TYPE E_Servo_State :
(
    DISABLED := 0,      // motor off
    ENABLING := 10,     // turning on
    HOME_NEEDED := 15,  // on but position unknown
    HOMING := 20,       // finding home
    READY := 30,        // ready for commands
    MOVING := 40,       // moving to target
    STOPPING := 45,     // slowing down
    ERRORED := 100,     // something wrong
    RESETTING := 110    // clearing errors
);
END_TYPE

(* stored: Version 1.1.0.1, ProductVersion 3.1.4024.13
   DUT E_Servo_State: Id {85c9793c-c72b-476c-98f8-1c1820b8b7bb} *)
